Pulse_length indicates on 3 outputs if an input pulse had been shorter than T_short (short = True), longer than T_long (long = True) or between T_short and T_long (middle = True).

*)
(* read system time *)
tx := TIME();

(* reset outputs, they should only be active 1 cycle *)
short := FALSE;
Middle := FALSE;
long := FALSE;

(* detect rising edge *)
IF in AND NOT edge THEN
	edge := TRUE;
	tn := tx;

(* detect for falling edge *)
ELSIF NOT in AND edge THEN
	edge := FALSE;
	tn := tx - tn;
	IF tn < t_short THEN
		short := TRUE;
	ELSIF tn > t_long THEN
		long := TRUE;
	ELSE
		Middle := TRUE;
	END_IF;

(* generate long pulse as soon as T_long is reached *)
ELSIF in AND tx - tn > t_long THEN
	long := TRUE;
END_IF;
END_FUNCTION_BLOCK

(* POU pwm_dc, ST *)
FUNCTION_BLOCK pwm_dc
VAR_INPUT
	F : REAL;
	DC : REAL;
END_VAR
VAR_OUTPUT
	Q : BOOL;
END_VAR
VAR
	clk: CLK_Prg;
	pulse: TP_R;
END_VAR

(*
	version 1.1	25 feb 2007
	programmer 	oscat
	tested BY		oscat

this signal generator generates a square wave signal which is specified by the frequency and the duty cycle
*)
CLK(PT := REAL_TO_TIME(1000/F));
Pulse(in := clk.Q, pt := REAL_TO_TIME(1000/F*DC));
Q := pulse.Q;

(* revision history

hm		25. feb 2007	rev 1.1
	recoded in st for better performance and better portability

*)
END_FUNCTION_BLOCK

(* POU TP_R, ST *)
FUNCTION_BLOCK TP_R
VAR_INPUT
	in : BOOL;
	PT : TIME;
END_VAR
VAR_OUTPUT
	Q : BOOL := 0;
	ET : TIME := t#0ms;
END_VAR
VAR
	edge : BOOL := FALSE;
	start : TIME := t#0ms;
END_VAR

(*
version 1.0	4 aug 2006
programmer 	hugo
tested by		tobias

retriggerable edge triggered pulse similar to TP but with a retrigger function
if the pt input is 0 then output is always low.
*)
(* rising edge trigger *)
IF in AND NOT edge THEN
	start := TIME();
	IF pt > t#0ms THEN Q := TRUE; END_IF;
END_IF;
edge := in;
IF q THEN
	et := TIME() - start;
	IF et >= PT THEN
		Q := FALSE;
		et := t#0ms;
	END_IF;
END_IF;
END_FUNCTION_BLOCK

(* POU pwm_pw, ST *)
FUNCTION_BLOCK pwm_pw
VAR_INPUT
	F : REAL;
	PW : TIME;
END_VAR
VAR_OUTPUT
	Q : BOOL;
END_VAR
VAR
	clk: CLK_Prg;
	pulse: TP_R;
END_VAR

(*
	version 1.1	25 feb 2007
	programmer 	oscat
	tested BY		oscat

this signal generator generates a square wave signal which is specified by the frequency and the pulse width.
*)
CLK(PT := REAL_TO_TIME(1000/F));
Pulse(in := clk.Q, pt := pw);
Q := pulse.Q;

(* revision history

hm		25. feb 2007	rev 1.1
	recoded in st for better performance and better portability

*)
END_FUNCTION_BLOCK

(* POU Real_To_StrF, ST *)
FUNCTION Real_To_StrF : STRING
VAR_INPUT
	IN : REAL;
	N : INT;
END_VAR
VAR
	dw1 : DWORD;
	dw2 : DWORD;
	s1: STRING;
	s2 : STRING;
END_VAR

(*
version 1.0	26 jan 2007
programmer 	hugo
tested by		tobias

Real_to_strF converts a Real to a fixed length String.
the string will be filles with leading zeroes to achieve the fixed length, or if too long, the lowest digits will be used.


*)
dw1 := TRUNC(ABS(in));
dw2 := TRUNC(round(fract(ABS(in))*EXPT(10,N),0));
IF in < 0 THEN
	s1 := CONCAT('-', DWORD_TO_STRING(dw1));
ELSE
	s1 := DWORD_TO_STRING(dw1);
END_IF;
	s1 := CONCAT(s1, '.');
s2 := DWORD_To_STRF(dw2,N);
Real_To_StrF := CONCAT(s1, s2);
END_FUNCTION

(* POU round, ST *)
FUNCTION round : REAL
VAR_INPUT
	in : REAL;
	N : INT;
END_VAR
VAR
END_VAR

(*
version 1.0	1 sep 2006
programmer 	hugo
tested by		tobias

this function rounds a real down to n digits behind the comma.
round(3.1415,1) = 3.1

*)
round := TRUNC(in * EXPT(10,N) + 0.5)/EXPT(10,N);
END_FUNCTION

(* POU Res_NI, ST *)
FUNCTION Res_NI : REAL
VAR_INPUT
	T : REAL;
	R0 : REAL;
END_VAR
VAR CONSTANT
	A : REAL := 0.5485;
	B : REAL := 0.665E-3;
	C : REAL := 2.805E-9;
END_VAR
VAR
END_VAR

(*
version 1.0	4 aug 2006
programmer 	hugo
tested by		tobias

this function returs the resistance for a nickel sensor for a temperature range from -60..+180 °C *)
Res_NI := R0 + A*T + B*EXPT(T,2) + C*EXPT(T,4);



(*

 Auszug aus DIN 43760 für Ni100

°C		R		°C		R		°C	R		°C		R		°C		R

-60 	69,5 	-10 	94,6 	40 	123,0 	90 		154,9 	140 	190,9
-55 	71,9 	-5 		97,3 	45 	126,0 	95 		158,3 	145 	194,8
-50 	74,3 	0 		100,0 	50 	129,1 	100 	161,8 	150 	198,7
-45 	76,7 	5 		102,8 	55 	132,2 	105 	165,3 	155 	202,6
-40 	79,1 	10 		105,6 	60 	135,3 	110 	168,8 	160 	206,6
-35 	81,6 	15 		108,4 	65 	138,5 	115 	172,4 	165 	210,7
-30 	84,2 	20 		111,2 	70 	141,7 	120 	176,0 	170 	214,8
-25 	86,7 	25 		114,1 	75 	145,0 	125 	179,6 	175 	219,0
-20 	89,3 	30 		117,1 	80 	148,3 	130 	183,3 	180 	223,2
-15 	91,9 	35 		120,0 	85 	151,6 	135 	187,1 	  	 

*)
END_FUNCTION

(* POU Res_PT, ST *)
FUNCTION Res_PT : REAL
VAR_INPUT
	T : REAL;
	R0 : REAL;
END_VAR
VAR CONSTANT
	A : REAL := 3.90802E-3 ;
	B : REAL := -5.802E-7;
	C : REAL := -4.27350E-12;
END_VAR
VAR
END_VAR

(*
version 1.1	4 Aug 2006
programmer 	hugo
tested by		tobias


this function returs the resistance for a platinum sensor for a temperature range from -200..+850 °C *)
IF T >= 0 THEN
	Res_PT := R0 * ( 1 + A*T + B*T*T);
ELSE
	Res_PT := R0 * ( 1 + A*T + B*T*T + C*(T-100)*T*T*T);
END_IF;


(*
 Auszug aus DIN 43760 für Pt100

°C		R		°C		R		°C	R			°C		R			°C		R			°C		R

-200 	18,49 	-100 	60,25 	0 	100,00 	100 	138,50 	200 	175,84 	300 	212,02
-195 	20,65 	-95 	62,28 	5 	101,95 	105 	140,39 	205 	177,68 	305 	213,80
-190 	22,80 	-90 	64,30 	10 	103,90 	110 	142,29 	210 	179,51 	310 	215,57
-185 	24,94 	-85 	66,31 	15 	105,85 	115 	144,17 	215 	181,34 	315 	217,35
-180 	27,08 	-80 	68,33 	20 	107,79 	120 	146,06 	220 	183,17 	320 	219,12
-175 	29,20 	-75 	70,33 	25 	109,73 	125 	147,94 	225 	184,99 	325 	220,88
-170 	31,32 	-70 	72,33 	30 	111,67 	130 	149,82 	230 	186,82 	330 	222,65
-165 	33,43 	-65 	74,33 	35 	113,61 	135 	151,70 	235 	188,63 	335 	224,41
-160 	35,33 	-60 	76,33 	40 	115,54 	140 	153,58 	240 	190,45 	340 	226,17
-155 	37,63 	-55 	78,32 	45 	117,47 	145 	155,45 	245 	192,26 	345 	227,92
-150 	39,71 	-50 	80,31 	50 	119,40 	150 	157,31 	250 	194,07 	350 	229,67
-145 	41,79 	-45 	82,29 	55 	121,32 	155 	159,18 	255 	195,88 	355 	231,42
-140 	43,87 	-40 	84,27 	60 	123,24 	160 	161,04 	260 	197,69 	360 	233,17
-135 	45,94 	-35 	86,25 	65 	125,16 	165 	162,90 	265 	199,49 	365 	234,91
-130 	48,00 	-30 	88,22 	70 	127,07 	170 	164,76 	270 	201,29 	370 	236,65
-125 	50,06 	-25 	90,19 	75 	128,98 	175 	166,61 	275 	203,08 	375 	238,39
-120 	52,11 	-20 	92,16 	80 	130,89 	180 	168,46 	280 	204,88 	380 	240,13
-115 	54,15 	-15 	94,12 	85 	132,80 	185 	170,31 	285 	206,67 	385 	241,86
-110 	56,19 	-10 	96,09 	90 	134,70 	190 	172,16 	290 	208,45 	390 	243,59
-105 	58,22 	-5 		98,04 	95 	136,60 	195 	174,00 	295 	210,24 	395 	245,31

*)
(*
revision history


*)
END_FUNCTION

(* POU Res_SI, ST *)
FUNCTION Res_SI : REAL
VAR_INPUT
	T : REAL;
	RS : REAL;
	TS : REAL;
END_VAR
VAR CONSTANT
	A : REAL := 7.64E-3;
	B : REAL := 1.66E-5;
END_VAR
VAR
END_VAR

(*
version 1.0	4 aug 2006
programmer 	hugo
tested by		tobias

this function returs the resistance for a silicon sensor for a temperature range from -50..+150 °C
for example KTY10 normaly Rs at 25 °C
*)
Res_SI := RS * ( 1 + A * (T - TS) + B * EXPT(T - TS, 2));
END_FUNCTION

(* POU rmp_B, ST *)
FUNCTION_BLOCK rmp_B
VAR_INPUT
	SET : BOOL := FALSE;
	PT : TIME;
	EN : BOOL := TRUE;
	UP : BOOL := TRUE;
	RST : BOOL := FALSE;
END_VAR
VAR_OUTPUT
	Out : BYTE := 0;
	busy: BOOL;
END_VAR
VAR
	last_step : TIME := T#0ms;
	now : TIME;
END_VAR

(*
	version 1.2	17 jan 2007
	programmer 	oscat
	tested BY		oscat

this ramp generator generates a byte wide ramp with 255 steps
the generator has an asynchronous set and reset
the ramp is controlled by PT which is the total ramp time for a full sweep from 0..255
an UD input controlls the direction Up or Down and the E input enables the ramp generation
a busy output indicates that the ramp is running, busy false means output is stable.

*)
IF en  THEN
	(* generate ramp *)
	now := TIME();
	IF now >= last_step + pt / 255 THEN
		last_step := now;
		IF UP AND out < 255 THEN out := out + 1; END_IF;
		IF NOT UP AND out > 0 THEN out := out -1; END_IF;
	END_IF;
END_IF;

(* check for asynchronous set or reset *)
IF set  THEN out := 255; END_IF;
IF rst THEN out := 0; END_IF;

(* checks for outputs stable and reset or set busy flag *)
IF out = 0 OR out = 255 THEN busy := FALSE; ELSE busy := TRUE; END_IF;

(* revision history

hm 5.10.2006	rev 1.1
	added busy output
hm 17.1.2007	rev 1.2
	renamed input ud to up for better usability
	deleted unused variable step

*)
END_FUNCTION_BLOCK

(* POU rmp_soft, ST *)
FUNCTION_BLOCK rmp_soft
VAR_INPUT
	IN : BOOL;
	val : BYTE;
END_VAR
VAR_INPUT CONSTANT
	pt_on: TIME := T#100ms;
	PT_off : TIME := T#100ms;
END_VAR
VAR CONSTANT
	steps : INT := 255;
END_VAR
VAR_OUTPUT
	Out : BYTE := 0;
END_VAR
VAR
	last_step : TIME := T#0ms;
	now : TIME;
	x :REAL := 0;
END_VAR

(*
	version 1.0	22 jan 2007
	programmer 	oscat
	tested BY		oscat

this soft on/off ramp generator generates a soft on and soft off ramp while the max on value is set by the input
the time for a full ramp can be set by config variables for up and down ramp.
*)
IF in  AND out < val THEN
	(* generate on ramp *)
	now := TIME();
	x := out + TIME_TO_REAL(now -last_step)*steps/TIME_TO_REAL(pt_on);
	IF x > val THEN
		out := val;
		x := val;
	ELSE out := REAL_TO_BYTE(x); END_IF;
	last_step := now;
ELSIF NOT in AND out > 0 THEN
	(* generate off ramp *)
	now := TIME();
	x := out - TIME_TO_REAL(now -last_step)*steps/TIME_TO_REAL(pt_off);
	IF x  < 0 THEN
		out := 0;
		x := 0;
	ELSE out := REAL_TO_BYTE(x); END_IF;
	last_step := now;
ELSIF in AND out > val THEN
	(* generate ramp down to input value *)
	now := TIME();
	x := out - TIME_TO_REAL(now -last_step)*steps/TIME_TO_REAL(pt_off);
	IF x  < val THEN
		out := val;
		x := val;
	ELSE out := REAL_TO_BYTE(x); END_IF;
	last_step := now;
END_IF;
IF out = val OR out = 0 THEN last_step := TIME(); END_IF;


(* revision history

hm 22.1.2007		rev 1.1
	deleted unused variables X1 and I, X2 and X3

*)
END_FUNCTION_BLOCK

(* POU rmp_W, ST *)
FUNCTION_BLOCK rmp_W
VAR_INPUT
	SET : BOOL := FALSE;
	PT : TIME;
	EN : BOOL := TRUE;
	UD : BOOL := TRUE;
	RST : BOOL := FALSE;
END_VAR
VAR_OUTPUT
	Out : WORD := 0;
	busy : BOOL;
END_VAR
VAR
	last_step : TIME := T#0ms;
	now : TIME;
END_VAR

(*
	version 1.2	22 Jan 2007
	programmer 	oscat
	tested BY		oscat

this ramp generator generates a Word wide ramp with 65535 steps
the generator has an asynchronous set and reset
the ramp is controlled by PT which is the total ramp time for a full sweep from 0..65535
an UD input controlls the direction Up or Down and the E input enables the ramp generation
a busy output indicates that the ramp is running, busy false means output is stable.
*)
IF en  THEN
	(* generate ramp *)
	now := TIME();
	IF now >= last_step + pt / 65535 THEN
		last_step := now;
		IF UD AND out < 65535 THEN out := out + 1; END_IF;
		IF NOT ud AND out > 0 THEN out := out -1; END_IF;
	END_IF;
END_IF;

(* check for asynchronous set or reset *)
IF set  THEN out := 65535; END_IF;
IF rst THEN out := 0; END_IF;

(* set or reset the busy flag *)
IF out = 0 OR out = 65535 THEN busy := FALSE; ELSE busy := TRUE; END_IF;

(* revision history:

hm 4.10.2006		rev 1.1
	added the busy output which signals that the ramp is running.

hm 22.1.2007		rev 1.2
	deleted unused variable step

*)
END_FUNCTION_BLOCK

(* POU scale_B2, ST *)
FUNCTION scale_B2 : REAL
VAR_INPUT
	in1: BYTE;
	in2: BYTE;
	K : REAL := 1;
	O : REAL := 0;
END_VAR
VAR_INPUT CONSTANT
	in1_min: REAL := 0;
	in1_max: REAL := 1000;
	in2_min: REAL := 0;
	in2_max: REAL := 1000;
END_VAR

(*
version 1.1	19 jan 2007
programmer 	hugo
tested by		tobias

	this functiob block can scale up to two inputs.
	the inputs have their min value at 0 and their max value at 255 while the min and max value can be either positive or negative.
	the inputs ramp between min and max values for the respective inputs to be between (0..255).
	the summed output is then scaled by an scale input K and a offset O can be added to the output.
	the min and max input configurations can be edited in the cfc editor by double clicking the symbol body.

*)
scale_B2 := 	((in1_max - in1_min)* in1 / 255 + in1_min +
				(in2_max - in2_min)* in2 / 255 + in2_min)
				* K + O;

(* revision History
hm 19.1.2007	rev 1.1
	changed outputs to real to avoid overflow of integer
	added offset for better cascading of scale functions
	changed from FB to function
*)
END_FUNCTION

(* POU scale_B4, ST *)
FUNCTION scale_B4 : REAL
VAR_INPUT
	in1: BYTE;
	in2: BYTE;
	in3: BYTE;
	in4: BYTE;
	K : REAL := 1;
	O : REAL := 0;
END_VAR
VAR_INPUT CONSTANT
	in1_min: REAL := 0;
	in1_max: REAL := 1000;
	in2_min: REAL := 0;
	in2_max: REAL := 1000;
	in3_min: REAL := 0;
	in3_max: REAL := 1000;
	in4_min: REAL := 0;
	in4_max: REAL := 1000;
END_VAR

(*
version 1.1	19 jan 2007
programmer 	hugo
tested by		tobias

	this functiob block can scale up to 4 inputs.
	the inputs have their min value at 0 and their max value at 255 while the min and max value can be either positive or negative.
	the inputs ramp between min and max values for the respective inputs to be between (0..255).
	the summed output is then scaled by an scale input K and a offset O can be added to the output.
	the min and max input configurations can be edited in the cfc editor by double clicking the symbol body.

*)
scale_B4 := 	((in1_max - in1_min)* in1 / 255 + in1_min +
				(in2_max - in2_min)* in2 / 255 + in2_min +
				(in3_max - in3_min)* in3 / 255 + in3_min +
				(in4_max - in4_min)* in4 / 255 + in4_min)
				* K + O;

(* revision History
hm 19.1.2007	rev 1.1
	changed outputs to real to avoid overflow of integer
	added offset for better cascading of scale functions
	changed from fb to function
*)
END_FUNCTION

(* POU scale_B8, ST *)
FUNCTION scale_B8 : REAL
VAR_INPUT
	in1: BYTE;
	in2: BYTE;
	in3: BYTE;
	in4: BYTE;
	in5: BYTE;
	in6: BYTE;
	in7: BYTE;
	in8: BYTE;
	K : REAL := 1;
	O : REAL := 0;
END_VAR
VAR_INPUT CONSTANT
	in1_min: REAL := 0;
	in1_max: REAL := 1000;
	in2_min: REAL := 0;
	in2_max: REAL := 1000;
	in3_min: REAL := 0;
	in3_max: REAL := 1000;
	in4_min: REAL := 0;
	in4_max: REAL := 1000;
	in5_min: REAL := 0;
	in5_max: REAL := 1000;
	in6_min: REAL := 0;
	in6_max: REAL := 1000;
	in7_min: REAL := 0;
	in7_max: REAL := 1000;
	in8_min: REAL := 0;
	in8_max: REAL := 1000;
END_VAR

(*
version 1.1	19 jan 2007
programmer 	hugo
tested by		tobias

	this functiob block can scale up to 8 inputs.
	the inputs have their min value at 0 and their max value at 255 while the min and max value can be either positive or negative.
	the inputs ramp between min and max values for the respective inputs to be between (0..255).
	the summed output is then scaled by an scale input K and a offset O can be added to the output.
	the min and max input configurations can be edited in the cfc editor by double clicking the symbol body.

*)
scale_B8 := 	((in1_max - in1_min)* in1 / 255 + in1_min +
				(in2_max - in2_min)* in2 / 255 + in2_min +
				(in3_max - in3_min)* in3 / 255 + in3_min +
				(in4_max - in4_min)* in4 / 255 + in4_min +
				(in5_max - in5_min)* in5 / 255 + in5_min +
				(in6_max - in6_min)* in6 / 255 + in6_min +
				(in7_max - in7_min)* in7 / 255 + in7_min +
				(in8_max - in8_min)* in8 / 255 + in8_min)
				* K + O;

(* revision History
hm 19.1.2007	rev 1.1
	changed outputs to real to avoid overflow of integer
	added offset for better cascading of scale functions
*)
END_FUNCTION

(* POU scale_X2, ST *)
FUNCTION scale_X2 : REAL
VAR_INPUT
	in1: BOOL;
	in2: BOOL;
	K : REAL := 1;
	O : REAL := 0;
END_VAR
VAR_INPUT CONSTANT
	in1_min: REAL := 0;
	in1_max: REAL := 1000;
	in2_min: REAL := 0;
	in2_max: REAL := 1000;
END_VAR

(*
version 1.0	19 jan 2007
programmer 	hugo
tested by		tobias

	this functiob block can scale up to two inputs.
	the input can select between two values with true or false.
	the summed output is then scaled by an scale input K and a offset O can be added to the output.
	the min and max input configurations can be edited in the cfc editor by double clicking the symbol body.

*)
IF NOT in1 THEN scale_x2 := in1_min; ELSE scale_x2 := in1_max; END_IF;
IF NOT in2 THEN scale_x2 := scale_x2 + in2_min; ELSE scale_x2 := scale_x2 + in2_max; END_IF;
scale_X2 := scale_X2 * k + O;

(* revision history

*)
END_FUNCTION

(* POU scale_X4, ST *)
FUNCTION scale_X4 : REAL
VAR_INPUT
	in1: BOOL;
	in2: BOOL;
	in3: BOOL;
	in4: BOOL;
	K : REAL := 1;
	O : REAL := 0;
END_VAR
VAR_INPUT CONSTANT
	in1_min: REAL := 0;
	in1_max: REAL := 1000;
	in2_min: REAL := 0;
	in2_max: REAL := 1000;
	in3_min: REAL := 0;
	in3_max: REAL := 1000;
	in4_min: REAL := 0;
	in4_max: REAL := 1000;
END_VAR

(*
version 1.0	19 jan 2007
programmer 	hugo
tested by		tobias

	this function can scale up to 4 inputs.
	the input can select between two values with true or false.
	the summed output is then scaled by an scale input K and a offset O can be added to the output.
	the min and max input configurations can be edited in the cfc editor by double clicking the symbol body.

*)
IF NOT in1 THEN scale_X4 := in1_min; ELSE scale_X4 := in1_max; END_IF;
IF NOT in2 THEN scale_x4 := scale_x4 + in2_min; ELSE scale_x4 := scale_x4 + in2_max; END_IF;
IF NOT in3 THEN scale_x4 := scale_x4 + in3_min; ELSE scale_x4 := scale_x4 + in3_max; END_IF;
IF NOT in4 THEN scale_x4 := scale_x4 + in4_min; ELSE scale_x4 := scale_x4 + in4_max; END_IF;
scale_X4 := scale_X4 * k + O;

(* revision history

*)
END_FUNCTION

(* POU scale_X8, ST *)
FUNCTION scale_X8 : REAL
VAR_INPUT
	in1: BOOL;
	in2: BOOL;
	in3: BOOL;
	in4: BOOL;
	in5: BOOL;
	in6: BOOL;
	in7: BOOL;
	in8: BOOL;
	K : REAL := 1;
	O : REAL := 0;
END_VAR
VAR_INPUT CONSTANT
	in1_min: REAL := 0;
	in1_max: REAL := 1000;
	in2_min: REAL := 0;
	in2_max: REAL := 1000;
	in3_min: REAL := 0;
	in3_max: REAL := 1000;
	in4_min: REAL := 0;
	in4_max: REAL := 1000;
	in5_min: REAL := 0;
	in5_max: REAL := 1000;
	in6_min: REAL := 0;
	in6_max: REAL := 1000;
	in7_min: REAL := 0;
	in7_max: REAL := 1000;
	in8_min: REAL := 0;
	in8_max: REAL := 1000;
END_VAR

(*
version 1.0	19 jan 2007
programmer 	hugo
tested by		tobias

	this function can scale up to 4 inputs.
	the input can select between two values with true or false.
	the summed output is then scaled by an scale input K and a offset O can be added to the output.
	the min and max input configurations can be edited in the cfc editor by double clicking the symbol body.

*)
IF NOT in1 THEN scale_x8 := in1_min; ELSE scale_x8 := in1_max; END_IF;
IF NOT in2 THEN scale_x8 := scale_x8 + in2_min; ELSE scale_x8 := scale_x8 + in2_max; END_IF;
IF NOT in3 THEN scale_x8 := scale_x8 + in3_min; ELSE scale_x8 := scale_x8 + in3_max; END_IF;
IF NOT in4 THEN scale_x8 := scale_x8 + in4_min; ELSE scale_x8 := scale_x8 + in4_max; END_IF;
IF NOT in5 THEN scale_x8 := scale_x8 + in5_min; ELSE scale_x8 := scale_x8 + in5_max; END_IF;
IF NOT in6 THEN scale_x8 := scale_x8 + in6_min; ELSE scale_x8 := scale_x8 + in6_max; END_IF;
IF NOT in7 THEN scale_x8 := scale_x8 + in7_min; ELSE scale_x8 := scale_x8 + in7_max; END_IF;
IF NOT in8 THEN scale_x8 := scale_x8 + in8_min; ELSE scale_x8 := scale_x8 + in8_max; END_IF;
scale_X8 := scale_X8 * k + O;

(* revision history

*)
END_FUNCTION

(* POU second_to_time, ST *)
FUNCTION second_to_time : TIME
VAR_INPUT
	input : REAL;
END_VAR
VAR
END_VAR

(*
version 1.0	4 aug 2006
programmer 	hugo
tested by		tobias

converts an amount of seconds in real to time
execution TIME on wago 750-841 =  17us 

*)
second_to_time := DWORD_TO_TIME(REAL_TO_DWORD(input * 1000));
END_FUNCTION

(* POU Sensor_Int, ST *)
FUNCTION Sensor_Int : REAL
VAR_INPUT
	Voltage : REAL;
	Current : REAL;
	RP : REAL;
	RS : REAL;
END_VAR
VAR
	Rx: REAL;
END_VAR

(*
version 1.1	20 jan 2007
programmer 	hugo
tested by		tobias

this function calculates the real resistance of a sensor RX given a parasitic resistor in parallel to the sensor and an additional serial resistor.
for example a parasitic parallel resistor for a PT100 can be ignored but a series resistor is the cable to the sensor.
for a humidity sensor, the parallel resistor is more dramatic and needs to be considered.
the function allows to consider a parallel and serial resistor at the same time.
with this function and known parasitic serial and parallel resistors the true resistance of the sensor can be calculated.

*)
Rx := RP * ( voltage / current - RS) / ( RP + RS - Voltage / Current);

(* revisaion history

hm 20.1.2007	rev 1.1
	deleted input R0 which was not needed.

*)
END_FUNCTION

(* POU sequence_4, ST *)
FUNCTION_BLOCK sequence_4
VAR_INPUT
	in0 : BOOL := TRUE;
	in1 : BOOL := TRUE;
	in2 : BOOL := TRUE;
	in3 : BOOL := TRUE;
	start : BOOL;
	rst : BOOL;
	wait0 : TIME := t#0s;
	delay0 : TIME := t#0s;
	wait1 : TIME := t#0s;
	delay1 : TIME := t#0s;
	wait2 : TIME := t#0s;
	delay2 : TIME := t#0s;
	wait3 : TIME := t#0s;
	delay3 : TIME := t#0s;
END_VAR
VAR_INPUT CONSTANT
	stop_on_error : BOOL := FALSE;
END_VAR
VAR_OUTPUT
	Q0 : BOOL;
	Q1 : BOOL;
	Q2 : BOOL;
	Q3 : BOOL;
	any : BOOL;
	run: BOOL;
	step : INT := -1;
	status : BYTE := 0;
END_VAR
VAR
	last : TIME;
	edge : BOOL;
	tx: TIME;
	init: BOOL;
END_VAR

(*
version 1.3	17 jan 2007
programmer 	oscat
tested by		hans

sequence_4 enables run when a low to high transition is present on start.
a low to high transition on start will restart the sequencer at any time while a rst will hold the sequencer in reset while true.
after run is enabled with a rising edge on start the sequencer waits for wait0 on in0 to enable q0 which stays on for delay0.
the next cycle starts with wait1, continues with delay 1 and so on...
if an edge is not detected during the wait period, the sequencer will then display the error number on the status output.
the status numbers 1..4 are errors in step 0..3.
after the last step that sets q3, the sequencer leaves q3 on for delay3 and then resets to the initial state.
a step output will indicate the current step of the sequencer and will also be present with a fault condition.
after the first output is turened on the sequencer switches from q0 to q1 and so on, at any time there is only one output enabled.
if an input signal is not detected during a wait period, the sequencer will display the error number ( 1 for in0, 2 for in1 .... ).
when an error is present and the config variable stop_on_error is set then the sequencer will stop. otherwise it will continue.
The status output will also display 110 for waiting and 111 for sequence running.
*)
(* read sps timer *)
tx := TIME();

(* initialize on startup *)
IF NOT init THEN
	last := tx;
	init := TRUE;
	status := 110;
END_IF;

(* asynchronous reset *)
IF rst THEN
	step := -1;
	Q0 := 0;
	Q1 := 0;
	Q2 := 0;
	Q3 := 0;
	status := 110;
	run := 0;

(* edge on start input restarts the sequencer *)
ELSIF start AND NOT edge THEN
	step := 0;
	last := tx;
	status := 111;
	Q0 := 0;
	Q1 := 0;
	Q2 := 0;
	Q3 := 0;
	run := 1;
END_IF;
edge := start;

(* check if stop on status is necessary *)
IF status > 0 AND status < 100 AND stop_on_error THEN RETURN; END_IF;

(* sequence is running *)
IF run AND step = 0 THEN
	IF NOT q0 AND in0 AND tx - last <= wait0 THEN
		Q0 := TRUE;
		last := tx;
	ELSIF NOT q0 AND tx - last > wait0 THEN
		status := 1;
		run := FALSE;
	ELSIF q0 AND tx - last >= delay0 THEN
		step := 1;
		last := tx;
	END_IF;
END_IF;
IF run AND step = 1 THEN
	IF NOT q1 AND in1 AND tx - last <= wait1 THEN
		Q0 := FALSE;
		Q1 := TRUE;
		last := tx;
	ELSIF NOT q1 AND Tx - last > wait1 THEN
		status := 2;
		q0 := FALSE;
		run := FALSE;
	ELSIF q1 AND tx - last >= delay1 THEN
		step := 2;
		last := tx;
	END_IF;
END_IF;
IF run AND step = 2 THEN
	IF NOT q2 AND in2 AND tx - last <= wait2 THEN
		Q1 := FALSE;
		Q2 := TRUE;
		last := tx;
	ELSIF NOT q2 AND Tx - last > wait2 THEN
		status := 3;
		q1 := FALSE;
		run := FALSE;
	ELSIF q2 AND tx - last >= delay2 THEN
		step := 3;
		last := tx;
	END_IF;
END_IF;
IF run AND step = 3 THEN
	IF NOT q3 AND in3 AND tx - last <= wait3 THEN
		Q2 := FALSE;
		Q3 := TRUE;
		last := tx;
	ELSIF NOT q3 AND Tx - last > wait3 THEN
		status := 4;
		q2 := FALSE;
		run := FALSE;
	ELSIF q3 AND tx - last >= delay3 THEN
		step := -1;
		q3 := FALSE;
		run := FALSE;
		status := 110;
	END_IF;
END_IF;
any := q0 OR q1 OR q2 OR q3;

(*
hm 1.10.06		rev 1.1
	corrected delay logic to be after event and not before
	added any output

hm 1.12.06		rev 1.2
	corrected failure in sequence logic.
	added init at startup to prevent from initial error after start.

hm 17.1.2007		rev 1.3
	changed output fault to status for better compatibility with other modules (ESR).
	added stop on error functionality and setup variable
	default for inputs in0..3 is true.
	renamed variable state to step
*)
END_FUNCTION_BLOCK

(* POU set_Tod, ST *)
FUNCTION set_Tod : TOD
VAR_INPUT
	hour : INT;
	minute : INT;
	second : REAL;
END_VAR
VAR
END_VAR

(*
version 1.0	4 aug 2006
programmer 	hugo
tested by		tobias

creates tod from hour minute and second 
execution time on wago 750-841 = 14 us  
*)
set_Tod := DWORD_TO_TOD(TRUNC(second * 1000) + minute * 60000 + hour * 3600000);
END_FUNCTION

(* POU SH, ST *)
FUNCTION_BLOCK SH
VAR_INPUT
	in : REAL;
	CLK : BOOL;
END_VAR
VAR_OUTPUT
	out : REAL;
	trig : BOOL;
END_VAR
VAR
	edge : BOOL;
END_VAR

(*
version 1.1	16 jan 2007
programmer 	hugo
tested by		tobias

this sample and hold module samples an input at the rising edge of clk an stores it in out.
the out stays stable until the next rising clk edge appears.
a trigger output as active for one cycle when the output was updated.

*)
IF clk AND NOT edge THEN
	out := in;
	trig := TRUE;
ELSE;
	trig := FALSE;
END_IF;
edge := clk;

(* revision history

hm 16.1.2007	rev 1.1
	added trig output

*)
END_FUNCTION_BLOCK

(* POU SH_1, ST *)
FUNCTION_BLOCK SH_1
VAR_INPUT
	in : REAL;
	PT : TIME;
END_VAR
VAR_OUTPUT
	out : REAL;
	Trig : BOOL;
END_VAR
VAR
	last : TIME;
END_VAR

(*
version 1.1	6 jan 2007
programmer 	hugo
tested by		tobias

this sample and hold module samples an input every PT seconds.
after a ample is taken the output Trig will be active for one cycle.

*)
IF TIME() - last >= PT THEN
	last := TIME();
	out := in;
	trig := TRUE;
ELSE
	trig := FALSE;
END_IF;

(* revision history

HM	6.1.2007	rev 1.1
	added trig output

*)
END_FUNCTION_BLOCK

(* POU SH_2, ST *)
FUNCTION_BLOCK SH_2
VAR_INPUT
	in : REAL;
	PT : TIME;
	N : INT;
	disc : INT;
END_VAR
VAR_OUTPUT
	out : REAL;
	trig : BOOL;
	avg : REAL;
	high: REAL;
	low: REAL;
END_VAR
VAR
	M : INT;
	buf : ARRAY[0..15] OF REAL;
	buf2 : ARRAY[0..15] OF REAL;
	last : TIME;
	i : INT;
	start: INT;
	temp: REAL;
	stop: INT;
END_VAR

(*
version 1.1	20 1 2007
programmer 	hugo
tested by		tobias

this sample and hold module samples an input every PT seconds.
this sample and hold also does avg and other calculations with the input data.
an average is calculated while for this calculation disc samples are discarded,
disc = 0 all samples are averaged,
if disc = 1 the lowest value is ignored,
if disc = 2 the lowest and highest values are ignored, 
and so on.....

*)
IF TIME() - last >= PT THEN
	last := TIME();
	trig := TRUE;

	(* limit M to 0..16 *)
	M := LIMIT(0,N,16);

	(* edge detected lets take the sample *)
	FOR i := M - 1 TO 1 BY -1 DO buf2[i] := buf2[i-1]; END_FOR;
	buf2[0] := in;
	out := in;
	buf := buf2;

	(* sort the ARRAY lowest value AT 0 *)
	FOR start := 0 TO M - 2 DO
		FOR i := start+1 TO M - 1 DO
			IF buf[start] > buf[i] THEN
				temp := buf[start];
				buf[start] := buf[i];
				buf[i] := temp;
			END_IF;
		END_FOR;
	END_FOR;

	(* any calculation with the samples is here *)
	stop := M - 1 - disc / 2;
	start := 0 + disc / 2;
	IF NOT even(disc) THEN start := start + 1; END_IF;
	avg := 0;
	FOR i := start TO stop DO avg := avg + buf[i]; END_FOR;
	avg := avg / (stop - start +1);
	low := buf[start];
	high := buf[stop];
ELSE
	Trig := FALSE;
END_IF;

(* revision history
hm 20.1.2007	rev 1.1
	added input N to specify the amout of samples for average and high low calculations
	added trig output

*)
END_FUNCTION_BLOCK

(* POU SH_T, ST *)
FUNCTION_BLOCK SH_T
VAR_INPUT
	in : REAL;
	EN : BOOL;
END_VAR
VAR_OUTPUT
	out : REAL;
END_VAR
VAR
END_VAR

(*
version 1.0	1 sep 2006
programmer 	hugo
tested by		tobias

this sample and hold module samples an input while en is high.
during the high time of en the output follows in.
the out stays stable until the en goes high again.
*)
IF en THEN out := in; END_IF;
END_FUNCTION_BLOCK

(* POU SHR_4E, ST *)
FUNCTION_BLOCK SHR_4E
VAR_INPUT
	SET : BOOL :=0;
	D0: BOOL := 0;
	CLK: BOOL;
	RST: BOOL :=0;
END_VAR
VAR_OUTPUT
	Q0: BOOL :=0;
	Q1: BOOL :=0;
	Q2: BOOL :=0;
	Q3: BOOL :=0;
END_VAR
VAR
	edge : BOOL :=1;
END_VAR

(*
version 1.0	4 aug 2006
programmer 	hugo
tested by		tobias

4 bit shift register with reset

executioin TIME on wago 750-841 =  8 us
*)
(* flankenerkennung clk wird high und edge war high reset ist nicht aktiv und set ist nicht aktiv *)
IF CLK AND edge AND NOT rst AND NOT set THEN
	edge := FALSE;	(* flanke wurde erkannt und weitere flankenerkennung wird verhindert bis edge wieder true ist *)
	(* hier ist der code für das ff aktivity *)
	Q3 := Q2;
	Q2 := Q1;
	Q1 := Q0;
	Q0 := D0;
END_IF
IF NOT clk THEN edge := TRUE; END_IF;	(* sobald clk wieder low wird warten auf nächste flanke *)
IF set AND NOT rst THEN						(* ausgang asynchron setzen wenn set aktiv und reset inaktiv. reset hat immer vorrang *)
	Q0 := TRUE;
	Q1 := TRUE;
	Q2 := TRUE;
	Q3 := TRUE;
END_IF;
IF rst THEN									(* wenn reset aktiv dann ausgang rücksetzen *)
	Q0 := FALSE;
	Q1 := FALSE;
	Q2 := FALSE;
	Q3 := FALSE;
END_IF;
END_FUNCTION_BLOCK

(* POU SHR_4UDE, ST *)
FUNCTION_BLOCK SHR_4UDE
VAR_INPUT
	set : BOOL :=0;
	D0: BOOL := 0;
	D3: BOOL := 0;
	CLK: BOOL;
	DN : BOOL :=0;
	RST: BOOL :=0;

END_VAR
VAR_OUTPUT
	Q0: BOOL :=0;
	Q1: BOOL :=0;
	Q2: BOOL :=0;
	Q3: BOOL :=0;
END_VAR
VAR
	edge : BOOL :=1;
END_VAR

(*
version 1.0	4 aug 2006
programmer 	hugo
tested by		tobias

4 bit shift register with reset up / down direction input

executioin TIME on wago 750-841 =  8 us
*)
(* flankenerkennung clk wird high und edge war high reset ist nicht aktiv und set ist nicht aktiv *)
IF CLK AND edge AND NOT rst AND NOT set THEN
	edge := FALSE;	(* flanke wurde erkannt und weitere flankenerkennung wird verhindert bis edge wieder true ist *)
	(* hier ist der code für das ff aktivity *)
	IF NOT dn THEN
		Q3 := Q2;
		Q2 := Q1;
		Q1 := Q0;
		Q0 := D0;
	ELSE
		Q0 := Q1;
		Q1 := Q2;
		Q2 := Q3;
		Q3 := D3;
	END_IF
END_IF
IF NOT clk THEN edge := TRUE; END_IF;	(* sobald clk wieder low wird warten auf nächste flanke *)
IF set AND NOT rst THEN						(* ausgang asynchron setzen wenn set aktiv und reset inaktiv. reset hat immer vorrang *)
	Q0 := TRUE;
	Q1 := TRUE;
	Q2 := TRUE;
	Q3 := TRUE;
END_IF;
IF rst THEN									(* wenn reset aktiv dann ausgang rücksetzen *)
	Q0 := FALSE;
	Q1 := FALSE;
	Q2 := FALSE;
	Q3 := FALSE;
END_IF;
END_FUNCTION_BLOCK

(* POU SHR_8PLE, ST *)
FUNCTION_BLOCK SHR_8PLE
VAR_INPUT
	Din : BOOL;
	Dload : BYTE;
	CLK: BOOL;
	UP: BOOL :=1;
	load : BOOL :=0;
	RST: BOOL :=0;
END_VAR
VAR_OUTPUT
	DOut: BOOL :=0;
END_VAR
VAR
	edge : BOOL :=1;
	register : BYTE := 0;
END_VAR

(*
version 1.0	4 aug 2006
programmer 	hugo
tested by		tobias

8 bit shift register with reset and parallel load
the register can shift up or down
it also has a serial input.
the Din input is on Bit0 for up shift and on bit 7 for down shift
the Dout output is on Bit7 for up shift and on bit 0 for down shift
paralle clock is performed clock synchron while a shift is performed first and then the register is reloaded

executioin TIME on wago 750-841 =  6 us
*)
(* flankenerkennung clk wird high und edge war high reset ist nicht aktiv und set ist nicht aktiv *)
IF CLK AND edge AND NOT rst THEN
	edge := FALSE;	(* flanke wurde erkannt und weitere flankenerkennung wird verhindert bis edge wieder true ist *)
	(* hier ist der code für das flankenevent *)
	IF UP THEN						(*shift up *)
		register := SHL(register,1);
		register.0 := Din;
		Dout := register.7;
	ELSE								(* shift down *);
		register := SHR(register,1);
		register.7 := Din;
		Dout := register.0;
	END_IF;
	IF load THEN							(* the byte on Din will be loaded if load = true *)
		register := Dload;
		IF up THEN Dout := register.7; ELSE Dout := register.0; END_IF;
	END_IF;
END_IF;
IF NOT clk THEN edge := TRUE; END_IF;	(* sobald clk wieder low wird warten auf nächste flanke *)
IF rst THEN									(* wenn reset aktiv dann ausgang rücksetzen *)
	register := 0;
	Dout := FALSE;
END_IF;
END_FUNCTION_BLOCK

(* POU SHR_8UDE, ST *)
FUNCTION_BLOCK SHR_8UDE
VAR_INPUT
	set : BOOL :=0;
	D0: BOOL := 0;
	D7: BOOL := 0;
	CLK: BOOL;
	DN : BOOL :=0;
	RST: BOOL :=0;
END_VAR
VAR_OUTPUT
	Q0: BOOL :=0;
	Q1: BOOL :=0;
	Q2: BOOL :=0;
	Q3: BOOL :=0;
	Q4: BOOL :=0;
	Q5: BOOL :=0;
	Q6: BOOL :=0;
	Q7: BOOL :=0;
END_VAR
VAR
	edge : BOOL :=1;
END_VAR

(*
version 1.0	4 aug 2006
programmer 	hugo
tested by		tobias

8 bit shift register with reset

executioin TIME on wago 750-841 =  8 us
*)
(* flankenerkennung clk wird high und edge war high reset ist nicht aktiv und set ist nicht aktiv *)
IF CLK AND edge AND NOT rst AND NOT set THEN
	edge := FALSE;	(* flanke wurde erkannt und weitere flankenerkennung wird verhindert bis edge wieder true ist *)
	(* hier ist der code für das ff aktivity *)
	IF NOT dn THEN
		Q7 := Q6;
		Q6 := Q5;
		Q5 := Q4;
		Q4 := Q3;
		Q3 := Q2;
		Q2 := Q1;
		Q1 := Q0;
		Q0 := D0;
	ELSE
		Q0 := Q1;
		Q1 := Q2;
		Q2 := Q3;
		Q3 := Q4;
		Q4 := Q5;
		Q5 := Q6;
		Q6 := Q7;
		Q7 := D7;
	END_IF
END_IF
IF NOT clk THEN edge := TRUE; END_IF;	(* sobald clk wieder low wird warten auf nächste flanke *)
IF set AND NOT rst THEN						(* ausgang asynchron setzen wenn set aktiv und reset inaktiv. reset hat immer vorrang *)
	Q0 := TRUE;
	Q1 := TRUE;
	Q2 := TRUE;
	Q3 := TRUE;
	Q4 := TRUE;
	Q5 := TRUE;
	Q6 := TRUE;
	Q7 := TRUE;
END_IF;
IF rst THEN									(* wenn reset aktiv dann ausgang rücksetzen *)
	Q0 := FALSE;
	Q1 := FALSE;
	Q2 := FALSE;
	Q3 := FALSE;
	Q4 := FALSE;
	Q5 := FALSE;
	Q6 := FALSE;
	Q7 := FALSE;
END_IF;
END_FUNCTION_BLOCK

(* POU sign_I, ST *)
FUNCTION sign_I : BOOL
VAR_INPUT
	in : INT;
END_VAR
VAR
END_VAR

(*
version 1.1	3 mar 2007
programmer 	hugo
tested by		tobias

this function return true if the integer input is negative

*)
IF in < 0 THEN
	sign_I := TRUE;
ELSE
	sign_I := FALSE;
END_IF;

(* revision history
hm 3.3.2007	rev 1.1
	changed method of function for better compatibility to other systems

*)
END_FUNCTION

(* POU sinH, ST *)
FUNCTION sinH : REAL
VAR_INPUT
	X : REAL;
END_VAR
VAR
END_VAR


(*
version 1.0	12 jan 2007
programmer 	hugo
tested by		tobias

this function calculates the sin hyperbolicus

*)
sinH := (EXPT(e,x) - EXPT(e,-x))/2;
END_FUNCTION

(* POU speed, ST *)
FUNCTION_BLOCK speed
VAR_INPUT
	ms : REAL;
	kmh : REAL;
	kn : REAL;
	mh : REAL;
END_VAR
VAR_OUTPUT
	Yms : REAL;
	Ykmh : REAL;
	Ykn : REAL;
	Ymh : REAL;
END_VAR
VAR
END_VAR

(*
version 1.0	27 mar 2007
programmer 	hugo
tested by		oscat

this function converts different speed units
any unused input can simply be left open.
different inputs connected at the same time will be added up.

*)
Yms := ms +
		kmh /3.6 +
		kn * 0.5144444 +
		mh * 0.44704;
Ykmh := Yms *3.6;
Ykn := Yms / 0.5144444;
Ymh := Yms / 0.44704;

(*
Geschwindigkeit Meter durch Sekunde m/s 1 m/s = 3,6 km/h
km durch (pro) Stunde, nicht „Stundenkilometer“ verwenden
Knoten kn 1 kn = 1 sm/h = 0,5144 m/s

*)
END_FUNCTION_BLOCK

(* POU sqrtn, ST *)
FUNCTION sqrtn : REAL
VAR_INPUT
	X : REAL;
	N : INT;
END_VAR
VAR
END_VAR

(*
version 1.0	12 jan 2007
programmer 	hugo
tested by		tobias

this function calculates the nth root function of X according to the formula sqrtn = x^(1/n).

*)
IF N > 1 THEN
	sqrtn := EXPT(x, 1.0 / INT_TO_REAL(n));
END_IF;
END_FUNCTION

(* POU STACK_16, ST *)
FUNCTION_BLOCK STACK_16
VAR_INPUT
	Din : DWORD;
	RW : BOOL;
	E : BOOL;
	RST : BOOL;
END_VAR
VAR_OUTPUT
	Dout : DWORD := 0;
	empty : BOOL := TRUE;
	full : BOOL := FALSE;
END_VAR
VAR
	Stack : ARRAY[0..15] OF DWORD;
	N : INT := -1;
	top : INT := 15;
END_VAR

(*
	version 1.0	4 aug 2006
	programmer 	hugo
	tested by		tobias

16 Dword STACK memory
*)
IF rst THEN
	(* asynchronous reset for the fifo *)
	N := -1;
	Dout := 0;
	empty := TRUE;
	full := FALSE;
ELSIF RW AND E AND NOT full THEN
	(* write action *)
	N := N + 1;
	IF N = top THEN full := TRUE; END_IF;
	empty := FALSE;
	stack[N] := Din;
ELSIF NOT RW AND E AND NOT empty THEN
	(* read from stack *)
	Dout := stack[N];
	N := N -1;
	IF N < 0 THEN empty := TRUE; END_IF;
	full := FALSE;
END_IF;
END_FUNCTION_BLOCK

(* POU STACK_32, ST *)
FUNCTION_BLOCK STACK_32
VAR_INPUT
	Din : DWORD;
	RW : BOOL;
	E : BOOL;
	RST : BOOL;
END_VAR
VAR_OUTPUT
	Dout : DWORD := 0;
	empty : BOOL := TRUE;
	full : BOOL := FALSE;
END_VAR
VAR
	Stack : ARRAY[0..31] OF DWORD;
	N : INT := -1;
	top : INT := 31;
END_VAR

(*
	version 1.0	4 aug 2006
	programmer 	hugo
	tested by		tobias

32 Dword STACK memory
*)
IF rst THEN
	(* asynchronous reset for the fifo *)
	N := -1;
	Dout := 0;
	empty := TRUE;
	full := FALSE;
ELSIF RW AND E AND NOT full THEN
	(* write action *)
	N := N + 1;
	IF N = top THEN full := TRUE; END_IF;
	empty := FALSE;
	stack[N] := Din;
ELSIF NOT RW AND E AND NOT empty THEN
	(* read from stack *)
	Dout := stack[N];
	N := N -1;
	IF N < 0 THEN empty := TRUE; END_IF;
	full := FALSE;
END_IF;
END_FUNCTION_BLOCK

(* POU stair, ST *)
FUNCTION stair : REAL
VAR_INPUT
	X : REAL;
	D : REAL;
END_VAR
VAR
	temp: REAL;
END_VAR


(*
version 1.0	28 jan 2007
programmer 	oscat
tested by		tobias

the function stair converts an anlog input signal to a staircase like output.
D is the step width for the output signal.
if D = 0 then the output follows the input without a chage.
*) 
temp := modR(X, D);
IF ABS(temp) < D / 2 THEN
	IF X > 0 THEN stair := X - temp; ELSE stair := X - temp; END_IF;
ELSE
	IF X > 0 THEN stair := X - temp + D; ELSE stair := X - temp - D; END_IF;
END_IF;
END_FUNCTION

(* POU stair2, ST *)
FUNCTION_BLOCK stair2
VAR_INPUT
	X : REAL;
	D : REAL;
END_VAR
VAR_OUTPUT
	Y: REAL;
END_VAR
VAR_TEMP
	tmp : REAL;
END_VAR


(*
version 1.0	28 jan 2007
programmer 	oscat
tested by		tobias

the function stair2 converts an anlog input signal to a staircase like output.
D is the step width for the output signal. the output will use D as a hysteresis for a stairchange.
if D = 0 then the output follows the input without a chage.
*) 
tmp := TRUNC(X / D);

IF X >= Y AND X >= 0 THEN
	Y := TRUNC(X / D) * D;
ELSIF X < Y AND X >= 0 THEN
	Y := (TRUNC(X/d) + 1) * D;
ELSIF X >= Y AND X < 0 THEN
	Y := (TRUNC(X/D)-1) * D;
ELSIF X < Y AND X < 0 THEN
	Y := TRUNC(X/D) *D;
END_IF;
END_FUNCTION_BLOCK

(* POU sun_pos, ST *)
FUNCTION_BLOCK sun_pos
VAR_INPUT
	latitude : REAL;				(* latitude of geographical position  *)
	longitude : REAL;				(* longitude of geographical position  *)
	utc : DT;						(*	world time				*)
END_VAR
VAR_OUTPUT
	B: REAL;
	HR: REAL;
END_VAR
VAR
	L: REAL;
	N: REAL; (* amount of days since 1.1.2000 12:00 *)
	G: REAL;
	K: REAL;
	A: REAL;
	X: REAL;
	D: REAL;
	JD: REAL;
	JD0: REAL;
	T: REAL;
	P: REAL;
	Ph: REAL;
	TA: REAL;
	H: REAL;
	RF: REAL;
	T1: REAL;
END_VAR

(*
version 1.0	1 Feb 2007
programmer 	hugo
tested by		tobias

this FUNCTION block calculates the sun position for a given date and time.
the times are calculated in utc and have to be corrected for the given time zone.
B is the angle from north and HR is the highth in degrees.

*)
N := (DT_TO_DWORD(utc) - 946728000)/86400.0;
JD := N + 2451545.0;
L := 280.460 + 0.9856474 * N;
L := modR(L,360);
G := 357.528 + 0.9856003 * N;
G := Rad(modR(G,360));
K := Rad(L + 1.915 * SIN(G) + 0.02 * SIN(2*G));
X := Rad(23.439 - 0.0000004 * N);
A := ATAN(COS(X)*SIN(K)/COS(K));
IF COS(K) < 0 THEN A := A + PI; END_IF;
D := ASIN(SIN(X) * SIN(K));
JD0 := TRUNC(JD - 0.5) + 0.5;
T := (TRUNC(N - 0.5) + 0.5) / 36525;
Ph := modR(6.697376 + 2400.05134 * T + 1.002738 * TOD_TO_REAL(DT_TO_TOD(utc))/3600000, 24);
P := PH * 15 + longitude;
TA := P - deg(A);
T1 := COS(Rad(TA))*SIN(Rad(latitude)) - TAN(D)*COS(Rad(latitude));
B := deg(ATAN(SIN(Rad(TA))/T1));
IF T1 < 0 THEN B := B + 180; END_IF;
IF B > 180 THEN
	B := B - 180;
ELSIF B < 180 THEN
	B := B + 180;
END_IF;
H := deg(ASIN(COS(D)*COS(Rad(TA))*COS(Rad(latitude))+SIN(D)*SIN(Rad(latitude))));
RF := 1.02 / TAN(Rad(H+10.3/(H+5.11)));
HR := H + RF / 60;
END_FUNCTION_BLOCK

(* POU sun_time, ST *)
FUNCTION_BLOCK sun_time
VAR_INPUT
	latitude : REAL;				(* latitude of geographical position  *)
	longitude : REAL;				(* longitude of geographical position  *)
	utc : DT;						(*	world time				*)
END_VAR
VAR_OUTPUT
	sun_midday : TOD;			(*	astrological midday in hours when sun stand at south direction	*)
	sun_rise : TOD;				(*	sun rise for current day in local time *)
	sun_set : TOD;				(*	sun set for current day in local time *)
	sun_declination : REAL;		(*	sun declination at midday in degrees	*)
END_VAR
VAR
	T: INT;							(* day in the year   *)
	DK: REAL;						(* sun declination at midday *)
	delta: REAL;					(* delta from midday for sunrise and sunset  *)
	h: REAL;
	B: REAL;
	offset : REAL;
END_VAR

(*
version 1.2	17 apr 2007
programmer 	hugo
tested by		tobias

this FUNCTION block calculates the sun rise, sun set, sun offset at midday sun declination for a given date 
for performance reasons the algorithm has been simplified and is accurate within a few minutes only 
the times are calculated in utc and have to be corrected for the given time zone
this correction is not done within sun_time because it would be a problem on days where dst is enabled or disabled

execution time on wago 750-841 is 30 us     
*)
B := Rad(latitude);
h := -0.0145;
T := day_of_year(DT_TO_DATE(utc));
offset := -0.1752 * SIN(0.033430*T + 0.5474) - 0.1340*SIN(0.018234*T - 0.1939);
sun_midday := hour_to_tod(12+Offset - longitude/15);
DK := 0.40954 * SIN(0.0172 * (T-79.35));
sun_declination := deg(DK);
delta := 12*ACOS((SIN(h) - SIN(B) * SIN(DK)) / (COS(B) * COS(DK)))/PI;
sun_rise := hour_to_tod(12 - delta - offset - longitude/15);
sun_set := hour_to_tod(12 + delta - Offset - longitude/15);

(* revision history

rev 1.1	hm	20.1.2007
	deleted unused variables sun_rineR and sun_setR

rev 1.2 hm 17.4.2007
	corrected error while sun:midday would not be corrected for longitude.
*)
END_FUNCTION_BLOCK

(* POU switch_I, ST *)
FUNCTION_BLOCK switch_I
VAR_INPUT
	set : BOOL;
	in : BOOL;
	rst : BOOL;
END_VAR
VAR_INPUT CONSTANT
	T_debounce : TIME := T#10ms;
	T_reconfig : TIME := T#1s;
	T_on_max : TIME := T#0h;
END_VAR
VAR_OUTPUT
	Q : BOOL := 0;
END_VAR
VAR
	state : BYTE := 0;
	edge : BOOL := 0;
	r_edge : BOOL := 0;
	T_on : TIME;
END_VAR

(*
version 1.0	4 aug 2006
programmer 	oscat
tested by		tobias

this is an intelligent switch interface which has an autodetect feature for in and it will detect the type of switch connected automatically
the input can be connected to low active pulses, high active pulses and on/off switch.
it will automatically adjust to the correct type without manual adjustment
a configurable debounce timer will debounce input signals
if t_on_max is set to anything other then 0 the output will be turned off after the max on time is reached.

*)
(* asynchronous set and reset first *)
IF set AND NOT rst THEN
	Q := 1;
	T_on := TIME();
ELSIF rst THEN
	Q := 0;
(* check FOR input edge AND start debounce timer *)
ELSIF (in XOR edge) AND NOT (state = 1) THEN
	state := 1;
	T_on := TIME();
(* edge was detected and debounce time elapsed *)
ELSIF (state = 1) AND (TIME() - t_debounce >= T_on) THEN
	state := 2;
	(* react on rising or falling edge depending on r_edge *)
	IF r_edge XOR in THEN Q := NOT Q; END_IF;
(* wait for T_reconfig and adjust r_edge *)
ELSIF state = 2 AND TIME() - t_reconfig >= T_on THEN
	r_edge := in;
END_IF;
IF Q AND T_on_max > t#0ms AND TIME() >= T_on + T_on_max THEN
	Q := FALSE;
END_IF;
edge := in;
END_FUNCTION_BLOCK

(* POU Switch_X, ST *)
FUNCTION_BLOCK Switch_X
VAR_INPUT
	IN1 : BOOL;
	IN2 : BOOL;
	IN3 : BOOL;
	IN4 : BOOL;
	IN5 : BOOL;
	IN6 : BOOL;
END_VAR
VAR_OUTPUT
	Q1 : BOOL;
	Q2 : BOOL;
	Q3 : BOOL;
	Q4 : BOOL;
	Q5 : BOOL;
	Q6 : BOOL;
	Q31 : BOOL;
	Q41 : BOOL;
	Q51 : BOOL;
	Q61 : BOOL;
	Q32 : BOOL;
	Q42 : BOOL;
	Q52 : BOOL;
	Q62 : BOOL;
END_VAR
VAR_INPUT CONSTANT
	t_debounce : TIME := t#50ms;
END_VAR
VAR
	init : BOOL;
	T1, T2, T3, T4, T5, T6 : TOF;
	tx: TIME;
	x1: BOOL;
	x2: BOOL;
	E1, E2 : BOOL;
END_VAR

(*
version 1.0	15 Feb 2007
programmer 	oscat
tested by		tobias

*)
(* initialize on startup *)
IF NOT init THEN
	init := TRUE;
	IF t_debounce < t#50ms THEN tx := t#50ms; ELSE tx := t_debounce; END_IF;
	T1(PT := Tx);
	T2(PT := Tx);
	T3(PT := Tx);
	T4(PT := Tx);
	T5(PT := Tx);
	T6(PT := Tx);
ELSE
	Q1 := FALSE;
	Q2 := FALSE;
	Q3 := FALSE;
	Q4 := FALSE;
	Q5 := FALSE;
	Q6 := FALSE;
	Q31 := FALSE;
	Q41 := FALSE;
	Q51 := FALSE;
	Q61 := FALSE;
	Q32 := FALSE;
	Q42 := FALSE;
	Q52 := FALSE;
	Q62 := FALSE;
END_IF;

(* read inputs and debounce *)
	T1(IN := IN1);
	T2(IN := IN2);
	T3(IN := IN3);
	T4(IN := IN4);
	T5(IN := IN5);
	T6(IN := IN6);

(* detect edge of IN1 and IN2 *)
IF t1.Q AND NOT E1 THEN X1 := TRUE; END_IF;
IF t2.Q AND NOT E2 THEN X2 := TRUE; END_IF;

IF t1.Q THEN
	IF t3.q THEN
		q31 := TRUE;
		X1 := FALSE;
	ELSIF t4.q THEN
		q41 := TRUE;
		X1 := FALSE;
	ELSIF t5.q THEN
		q51 := TRUE;
		X1 := FALSE;
	ELSIF t6.q THEN
		q61 := TRUE;
		X1 := FALSE;
	END_IF;
ELSIF t2.Q THEN
	IF t3.q THEN
		q32 := TRUE;
		X2 := FALSE;
	ELSIF t4.q THEN
		q42 := TRUE;
		X2 := FALSE;
	ELSIF t5.q THEN
		q52 := TRUE;
		X2 := FALSE;
	ELSIF t6.q THEN
		q62 := TRUE;
		X2 := FALSE;
	END_IF;
(* in1 was active alone *)
ELSIF NOT T1.Q AND E1 AND X1 THEN
	Q1 := TRUE;
	X1 := FALSE;
ELSIF NOT T2.Q AND E2 AND X2 THEN
	Q2 := TRUE;
	X2 := FALSE;
ELSIF T3.Q THEN
	Q3 := TRUE;
ELSIF T4.Q THEN
	Q4 := TRUE;
ELSIF T5.Q THEN
	Q5 := TRUE;
ELSIF T6.Q THEN
	Q6 := TRUE;
END_IF;

(* save state of in1 and in2 *)
E1 := T1.Q;
E2 := T2.Q;
END_FUNCTION_BLOCK

(* POU tanH, ST *)
FUNCTION tanH : REAL
VAR_INPUT
	X : REAL;
END_VAR
VAR
END_VAR


(*
version 1.0	12 jan 2007
programmer 	hugo
tested by		tobias

this function calculates the tangens hyperbolicus

*)
tanH := -2 / (EXPT(e, -2 * x) + 1) + 1;
END_FUNCTION

(* POU temp_ext, ST *)
FUNCTION_BLOCK temp_ext
VAR_INPUT
	t_ext1 : REAL;
	t_ext2 : REAL;
	t_ext3 : REAL;
	t_ext_config : BYTE := 0;
	dt_in : DT;
END_VAR
VAR_INPUT CONSTANT
	t_ext_min : REAL := -40;
	t_ext_max : REAL := 60;
	t_ext_default : REAL := -10;
	heat_period_start : DATE := D#1970-9-1;
	heat_period_stop : DATE := D#1970-4-30;
	cool_period_start : DATE := D#1970-4-1;
	cool_period_stop : DATE := D#1970-9-30;
	heat_start_temp_day : REAL := 15;
	heat_start_temp_night : REAL := 10;
	heat_stop_temp : REAL := 18;
	cool_start_temp_day : REAL := 26;
	cool_start_temp_night : REAL := 26;
	cool_stop_temp : REAL := 24;
	start_day : TOD := tod#09:00;
	start_night : TOD := tod#21:00;
	cycle_time : TIME := t#10m;
END_VAR
VAR_OUTPUT
	t_ext : REAL;
	heat : BOOL;
	cool : BOOL;
END_VAR
VAR
	tx: TIME;
	last_run: TIME;
	init: BOOL;
	cool_start: DATE;
	cool_stop: DATE;
	heat_start: DATE;
	heat_stop: DATE;
	xdate: DATE;
	day: BOOL;
END_VAR


(*
version 1.0	6 dec 2006
programmer 	hugo
tested by		tobias

temp_ext measures and processes ext temperature and decides if heating or cooling is needed.

 the measurement of t_ext has 3 inputs which can be configured in different ways:
	t_ext_config = 0 means the ext temp is the avg of the 3 external temperatures, this mode is the default mode.
	t_ext_config = 1 means t_ext1 is used.
	t_ext_config = 2 means t_ext1 is used.
	t_ext_config = 3 means t_ext1 is used.
	t_ext_config = 4 means t_ext_default is used.
	t_ext_config = 5 means the lowest of the 3 external temperatures is used.
	t_ext_config = 6 means the higest externnal temperature is used.
	t_ext_config = 7 means the midlle external temperature is used, if there are only two working, the lowest is used.
	in any config mode, an external temperature higher then t_ext_max or lower then t_ext_min is ignored to prevent from temperatures caused by broken sensors or wires.
	if no external temperature is available, a default value (t_ext_default) is used.
	if you have only one external sensor, connect the 3 inputs to the same sensor, or select the right input with t_ext_config.

heating or cooling is enabled during heating / cooling period when the day or night start temperature is reached for at least the specified delay time and will be disabled after the stop temperature is reached. 
t_ext output can be used by other modules to determine the correct system temperature for heating or cooling.

*)
IF NOT init THEN
	init := TRUE;
	heat_start := set_Date(1972,month(heat_period_start),day_of_month(heat_period_start));
	heat_stop := set_Date(1972,month(heat_period_stop),day_of_month(heat_period_stop));
	cool_start := set_Date(1972,month(cool_period_start),day_of_month(cool_period_start));
	cool_stop := set_Date(1972,month(cool_period_stop),day_of_month(cool_period_stop));
END_IF;
tx := TIME();

(* for efficiency exit isf this program has been executed less then 1min ago *)
IF tx - last_run < cycle_time THEN RETURN; END_IF;

(* calculate frequently used variables *)
xdate := set_Date(1972,month(DT_TO_DATE(dt_in)),day_of_month(DT_TO_DATE(dt_in)));
day := DT_TO_TOD(dt_in) >= start_day AND  DT_TO_TOD(dt_in) < start_night;

(* read the correct external temperature depending on the t_ext_config setting *)
t_ext := multi_in(t_ext1, t_ext2, t_ext3, t_ext_default, t_ext_min, t_ext_max, t_ext_config);

(* dtermine heating *)
IF (heat_start <= heat_stop AND xdate >= heat_start AND xdate <= heat_stop) OR (heat_start > heat_stop AND (xdate >= heat_start OR xdate <= heat_stop)) THEN
	(* heating period id true check for temperature *)
	IF day AND t_ext <= heat_start_temp_day THEN
		heat := TRUE;
	ELSIF NOT day AND t_ext <= heat_start_temp_night THEN
		heat := TRUE;
	ELSIF t_ext >= heat_stop_temp THEN
		heat := FALSE;
	END_IF;
ELSE
	heat := FALSE;
END_IF;

(* dtermine cooling *)
IF (cool_start <= cool_stop AND xdate >= cool_start AND xdate <= cool_stop) OR (cool_start > cool_stop AND (xdate >= cool_start OR xdate <= cool_stop)) THEN
	(* cooling period is true check for temperature *)
	IF day AND t_ext >= cool_start_temp_day THEN
		cool := TRUE;
	ELSIF NOT day AND t_ext >= cool_start_temp_night THEN
		cool := TRUE;
	ELSIF t_ext <= cool_stop_temp THEN
		cool := FALSE;
	END_IF;
ELSE
	cool := FALSE;
END_IF;

last_run := tx;
END_FUNCTION_BLOCK

(* POU Temp_NI, ST *)
FUNCTION Temp_NI : REAL
VAR_INPUT
	Res : REAL;
	R0 : REAL;
END_VAR
VAR CONSTANT
	accuracy: REAL := 0.001;
END_VAR
VAR
	step: REAL;
END_VAR

(*
version 1.1	24 jan 2007
programmer 	hugo
tested by		tobias

this function returs the temperature for a nickel sensor for a range from -60..+180 °C *)
(* since the formula cannot be solved this is a successive approximation *)
Temp_NI := -60;
step := 120;
WHILE step > accuracy DO
	(* test if result greater or less *)
	IF Res_NI(Temp_NI + step,R0) < res THEN Temp_NI := Temp_NI + step; END_IF;
	step := step / 2;
END_WHILE;


(* revision history

hm 24.1.2007	deleted unused variable A, B, C

*)
END_FUNCTION

(* POU Temp_PT, ST *)
FUNCTION Temp_PT : REAL
VAR_INPUT
	Res : REAL;
	R0 : REAL;
END_VAR
VAR CONSTANT
	A : REAL := 3.9083E-3 ;
	B : REAL := -5.775E-7;
	accuracy : REAL := 0.001;
END_VAR
VAR
	step: REAL;
END_VAR

(*
version 1.1	24 jan 2007
programmer 	hugo
tested by		tobias

this function returs the temperature for a platinum sensor for a range from -200..+850 °C *)
IF Res >= R0 THEN
	Temp_PT := (-A*R0 + SQRT(EXPT(A*R0,2) - 4*B*R0 * (R0-Res))) / (2 * B * R0);
ELSE
	(* since the formula cannot be solved this is a successive approximation *)
	Temp_PT := -200;
	step := 100;
	WHILE step > accuracy DO
		(* test if result greater or less *)
		IF Res_PT(Temp_PT + step,R0) < res THEN Temp_PT := Temp_PT + step; END_IF;
		step := step / 2;
	END_WHILE;
END_IF;

(* revision history

hm 24.1.2007	deleted unused variable C

*)
END_FUNCTION

(* POU Temp_SI, ST *)
FUNCTION Temp_SI : REAL
VAR_INPUT
	Res : REAL;
	RS : REAL;
	TS : REAL;
END_VAR
VAR CONSTANT
	A : REAL := 7.64E-3;
	B : REAL := 1.66E-5;
END_VAR
VAR
END_VAR

(*
version 1.1	24 jan 2007
programmer 	hugo
tested by		tobias

this function returs the temperature for a silicon sensor for a range from -50..+150 °C
for example KTY10 RS at TS normally 25 °C
*)
Temp_SI := TS + (SQRT(EXPT(A,2) - 4 * B * ( 1 -  Res / RS ) - A) / ( 2 * B));


(* revision history

hm 24.1.2007		rev 1.1
the function would only word for TS = 25, now it works for other values of ts.


*)
END_FUNCTION

(* POU timer_2, ST *)
FUNCTION_BLOCK timer_2
VAR_INPUT
	DT_in : DT;
	start : TOD;
	duration : TIME;
	mode : BYTE;
	holiday : BOOL;
END_VAR
VAR_OUTPUT
	Q : BOOL;
END_VAR
VAR
	last_check : TIME := T#0s;
	dat : DATE;
	daytime : TOD;
	activation: TIME;
	tx: TIME;
	enabled: BOOL;
	wday: INT;
	init: BOOL;
END_VAR

VAR RETAIN
	run_date : DATE;
END_VAR

(*
version 1.1	22 Feb 2007
programmer 	oscat
tested by		tobias

this timer generated programmabe output pulses per day, week, month and so on.
the mode input determines on which days the timer will be active.
	mode = 0			never
	mode = 1..7		monday .. sunday
	mode = 11			every day
	mode = 12			every second day
	mode = 13			every 3rd day
	mode = 14			every 4th day
	mode = 15			every 5th day
	mode = 16 		every 6th day
	mode = 20			only monday - friday
	mode = 21			only sat - sunday
	mode = 22			workdays only
	mode = 23			holidays and weekend
	mode = 24			holidays only
	mode = 25			every 1st day of the month
	mode = 26			every last day of the month
	mode = 27			every 31 of december
	mode = 28			every 1st of january

a holiday input can be used to supply holiday information to the module.
*)
tx := TIME();

IF NOT init THEN
	init := TRUE;
	last_check := tx - t#100ms;
END_IF;

(* for performance resons exit if execution is not necessary *)
IF tx - last_check <= T#100ms THEN RETURN; END_IF;

(* calculate temp variables *)
dat := DT_TO_DATE(dt_in);
daytime := DT_TO_TOD(dt_in);
wday := weekday(dat);

(* calculate if any action is necessary today *)
enabled := FALSE;
CASE mode OF
1..7:	(* mondays to fridays *)
	IF wday = mode THEN enabled := 1; END_IF;
11:	(* every day *)
	enabled := TRUE;
12..16:	(* every nth day *)
	IF (TRUNC(DATE_TO_DWORD(dat)/86400)) MOD (mode - 10) = 0 THEN enabled := 1; END_IF;
20:	(* monday - friday *)
	IF wday <= 5 THEN enabled := TRUE; END_IF;
21:	(* saturday and sunday *)
	IF wday > 5 THEN enabled := TRUE; END_IF;
22: (* workdays only *)
	IF wday <= 5 AND NOT holiday THEN enabled := TRUE; END_IF;
23:	(* holidays and weekends *)
	IF wday > 5 OR holiday THEN enabled := TRUE; END_IF;
24:	(* holidays only *)
	enabled := holiday;
25:	(* 1st day of the month *)
	IF day_of_month(dat) = 1 THEN enabled := TRUE; END_IF;
26:	(* last day of month *)
	IF day_of_month(dat + t#1d) = 1 THEN enabled := TRUE; END_IF;
27:	(* 31st of december *)
	IF day_of_month(dat) = 31 AND month(dat) = 12 THEN enabled := TRUE; END_IF;
28:	(* 1st of january *)
	IF day_of_year(dat) = 1 THEN enabled := TRUE; END_IF;
END_CASE;

(* set or reset output if necessary *)
IF enabled AND NOT Q AND daytime >= start AND run_date <> dat THEN
	Q := 1;
	activation := tx;
	run_date := dat;
ELSIF Q AND tx - activation >= duration THEN
	Q := 0;
END_IF;
last_check := Tx;


(* revision history
hm 22.2.2007		rev 1.1
	changed VAR RETAIN PERSISTENT to VAR RETAIN for better compatibility
	wago lon contollers do not support persisitent

*)
END_FUNCTION_BLOCK

(* POU WCT, ST *)
FUNCTION WCT : REAL
VAR_INPUT
	T : REAL;
	V : REAL;
END_VAR
VAR
END_VAR

(*
version 1.0	7 Feb 2007
programmer 	hugo
tested by		tobias

this function calculates the wind chill temperature

*)
IF V < 5 OR T > 10 THEN
	WCT := T;
ELSE
	WCT := 13.12 + 0.6215 * T +(0.3965 * T - 11.37) * EXPT(v, 0.16);
END_IF;
END_FUNCTION

(* POU window, ST *)
FUNCTION window : BOOL
VAR_INPUT
	low : REAL;
	in : REAL;
	high : REAL;
END_VAR
VAR
END_VAR

(*
	version 1.1	22 jan 2007
	programmer 	hugo
	tested BY		tobias

this checks a signal if the signal is between the upper and lower limit
*)
window := in < high AND in > low;


(* revision history
hm	22.1.2007	rev 1.1
	changed the order of inputs to low, in, high

*)
END_FUNCTION

(* POU Word_of_Byte, ST *)
FUNCTION Word_of_Byte : WORD
VAR_INPUT
	B0 : BYTE;
	B1 : BYTE;
END_VAR
VAR
END_VAR

(*
version 1.0	24 jan 2007
programmer 	hugo
tested by		tobias

this function creates a word from 2 individual bytes

*)
Word_of_Byte := B1;
Word_of_Byte := SHL(Word_of_Byte,8) + B0;
END_FUNCTION

(* POU Word_of_Dword, ST *)
FUNCTION Word_of_Dword : WORD
VAR_INPUT
	in : DWORD;
	N : BYTE;
END_VAR
VAR
	temp: DWORD;
END_VAR

(*
version 1.0	17 jan 2007
programmer 	hugo
tested by		tobias

this function extracts a single word from the nth position from right (right is lowest byte)
the lower word (starting weith Bit0 from in) is selected with N=0.
*)
temp := SHR(in,n*16);
Word_of_Dword := DWORD_TO_WORD(temp);
END_FUNCTION

(* POU work_week, ST *)
FUNCTION work_week : INT
VAR_INPUT
	idate : DATE;
END_VAR
VAR
	wday1 : INT;
END_VAR

(*
version 1.1	14 jan 2007
programmer 	hugo
tested by		tobias

calculates the work week for a given date  
execution time on wago 750-841 = 155us   
*)
wday1 := weekday(set_Date(year(idate), 1,1));
IF wday1 < 5 THEN
	work_week := TRUNC((day_of_year(idate) + wday1 + 5)/7); ELSE
	work_week := TRUNC((day_of_year(idate) + wday1 - 2)/7); END_IF


(* revision history

hm 17.1.2007		rev 1.1
	deleted unused variable yday

*)
END_FUNCTION
